FUNCTION_BLOCK PUBLIC FB_SerialCommunicationCluster
VAR	
	fbSerialCommunication01		: FB_SerialCommunication(nDatabits := nInternalDatabits, eParity := eInternalParity, nStopbits := nInternalStopbits);
	fbSerialCommunication02		: FB_SerialCommunication(nDatabits := nInternalDatabits, eParity := eInternalParity, nStopbits := nInternalStopbits);
	nInternalDatabits    		: BYTE(7..8);
	eInternalParity         	: E_Parity;
	nInternalStopbits			: BYTE(1..2);
END_VAR

fbSerialCommunication01();
fbSerialCommunication02();

METHOD FB_init : BOOL
VAR_INPUT
	bInitRetains	: BOOL; // if TRUE, the retain variables are initialized (warm start / cold start)
	bInCopyCode		: BOOL; // if TRUE, the instance afterwards gets moved into the copy code (online change)
	nDatabits    	: BYTE(7..8);
	eParity         : E_Parity;
	nStopbits		: BYTE(1..2);	
END_VAR
fbSerialCommunication01.FB_init(bInitRetains := bInitRetains, bInCopyCode := bInCopyCode, nDatabits := nDatabits, eParity := eParity, nStopbits := nStopbits);
fbSerialCommunication02.FB_init(bInitRetains := bInitRetains, bInCopyCode := bInCopyCode, nDatabits := nDatabits, eParity := eParity, nStopbits := nStopbits);

THIS^.nInternalDatabits := nDatabits;
THIS^.eInternalParity := eParity;
THIS^.nInternalStopbits := nStopbits;
END_METHOD

END_FUNCTION_BLOCK

(* stored: Version 1.1.0.1, ProductVersion 3.1.4022.18
   POU FB_SerialCommunicationCluster: Id {c650a89b-d82e-4f8e-97d4-08dc50d14f44}, SpecialFunc None
   Method FB_init: Id {c7d7699e-e136-4a46-8854-c8bc3bf114a6} *)
